FUNCTION_BLOCK FB_ATMTest EXTENDS FB_TestSuite
VAR
    (* Caller-owned axis, persistent storage, and Y motor.
       In a real PRG the AxisRef would come from MAIN.Mxx. *)
    axRef    : AXIS_REF;
    fbPDS    : LCLS_Tc_DevAbs.FB_PersistentDataStorage;

    (* FB_ATM is single-axis (nActiveMotorCount := 1), so only slot 1
       holds a real motor. aiMotionStage is sized to
       MotionConstants.MAX_STATE_MOTORS to match FB_ATM.FB_Init's
       fixed-size signature; slots 2-4 default-init to a nil interface
       and are never touched. *)
    fbMotorY : FB_MotionStageNC(AxisRef := axRef, iPersistentDataStorage := fbPDS, sName := 'Y');
    aiMotionStage : ARRAY[1..MotionConstants.MAX_STATE_MOTORS] OF I_MotionStage := [fbMotorY];

    {attribute 'pytmc' := '
        pv: MMS
        astPositionState.array: 1..6
    '}
    astPositionState : ARRAY[1..MotionConstants.MAX_STATE_MOTORS]
                         OF ARRAY[1..GeneralConstants.MAX_STATES] OF ST_PositionState;

    fbFFHWO    : FB_HardwareFFOutput;
    fbArbiter  : FB_Arbiter(1);
    fbSubSysIO : FB_DummyArbIO;

    sDeviceName    : STRING := 'TST:ATM';
    sTransitionKey : STRING := 'TST:ATM-TRANSITION';

    fbATM : FB_ATM(
        aiMotionStage         := aiMotionStage,
        astPositionState      := astPositionState,
        fbFFHWO               := fbFFHWO,
        fbArbiter             := fbArbiter,
        sDeviceName           := sDeviceName,
        sTransitionKey        := sTransitionKey,
        bEnableBeamParams     := TRUE,
        bEnablePositionLimits := TRUE,
        bReadDBNow            := TRUE
    );

    (* Per-install PMPS-side state config (caller-owned). Mirrors what
       a real PRG_xxL0_ATM would declare. stDefault is the caller-owned
       baseline template that FB_CC_StatePMPSConfig's inner FB_StateSetup
       preloads from; fbATM subsequently overrides per-state sName and
       fDelta via its own FB_CC_DeviceStateDefaults array. *)
    stDefault : ST_PositionState := (
        bMoveOk       := TRUE,
        bValid        := TRUE,
        bUseRawCounts := FALSE
    );

    afbStatePMPS : ARRAY[1..6] OF FB_CC_StatePMPSConfig[
        (stPositionState := astPositionState[1][E_ATM_States.OUT],
         stDefault       := stDefault,
         fPosition       := 10,
         sPmpsState      := 'TST:ATM-OUT'),
        (stPositionState := astPositionState[1][E_ATM_States.TARGET1],
         stDefault       := stDefault,
         fPosition       := 20,
         sPmpsState      := 'TST:ATM-TARGET1'),
        (stPositionState := astPositionState[1][E_ATM_States.TARGET2],
         stDefault       := stDefault,
         fPosition       := 30,
         sPmpsState      := 'TST:ATM-TARGET2'),
        (stPositionState := astPositionState[1][E_ATM_States.TARGET3],
         stDefault       := stDefault,
         fPosition       := 40,
         sPmpsState      := 'TST:ATM-TARGET3'),
        (stPositionState := astPositionState[1][E_ATM_States.TARGET4],
         stDefault       := stDefault,
         fPosition       := 50,
         sPmpsState      := 'TST:ATM-TARGET4'),
        (stPositionState := astPositionState[1][E_ATM_States.TARGET5],
         stDefault       := stDefault,
         fPosition       := 60,
         sPmpsState      := 'TST:ATM-TARGET5')
    ];

    bFirstScan : BOOL := TRUE;
    i          : UINT;
END_VAR

(* Fake PMPS handling. *)
fbSubSysIO(
    LA  := fbArbiter,
    FFO := fbFFHWO
);

(* Caller-side PMPS configurators write each slot once in
   FB_CC_StatePMPSConfig.CallAfterInit; no cyclic tick. *)

(* One-shot motor setup + initial caller-owned enables. Limits,
   brake/enable modes, home cmd, user/hardware enables, default
   velocity; skip NC param restore. *)
IF bFirstScan THEN
    fbMotorY.SetModeEnableLimits(
        LimBackward    := TRUE,
        LimForward     := TRUE,
        HomeEnable     := FALSE,
        BrakeMode      := E_StageBrakeMode.IF_ENABLED,
        EnableMode     := E_StageEnableMode.DURING_MOTION,
        HomeMode       := E_EpicsHomeCmd.LOW_LIMIT,
        UserEnable     := TRUE,
        HardwareEnable := TRUE
    );
    fbMotorY.SetVelocity(Velocity := 15.5);
    fbMotorY.RestoreMotionParams      := FALSE;
    fbMotorY.DoNotRestoreNcParameters := TRUE;

    bFirstScan := FALSE;
END_IF

fbPDS();
fbMotorY();
fbATM();

TestStateMove();
TestTempFFO();

METHOD SetATMTemp
VAR_INPUT
    iTempC : INT;
END_VAR
VAR
    ptr : POINTER TO INT;
END_VAR
ptr  := ADR(fbATM.fbTempSensor1.iRaw);
ptr^ := iTempC * 10;
END_METHOD

(*
    Smoke test for ATM state-move wiring. Walks OUT then TARGET1 and
    asserts each lands within fTolerance of the configured fPosition.
    Mirrors FB_REFTest: stageReady gate up front, NOT bMoving +
    position-tolerance check per state, 60s watchdog, on timeout
    AssertTrue(FALSE, ...) with the current step and observed
    position. Two moves is enough to exercise the FB wiring; the
    motion stack itself is covered by the
    lcls-twincat-motion-abstraction test suite.
*)
METHOD TestStateMove
VAR_INST
    tonTimer  : TON;
    nTestStep : INT := 0;
    fObserved : LREAL;
END_VAR
VAR CONSTANT
    fTolerance : LREAL := 2.0;
END_VAR
TEST('TestATMStateMove');

tonTimer(IN := TRUE, PT := T#60s);
fObserved := fbMotorY.stMotionStatus.fActPosition;

CASE nTestStep OF
    0:
        IF fbMotorY.stMotionStatus.bStageReady
           AND NOT fbMotorY.stMotionStatus.bError THEN
            fbATM.eEnumSet := E_ATM_States.OUT;
            nTestStep      := 1;
        END_IF
    1:
        (* OUT is configured at fPosition := 10 in afbStatePMPS[1]. *)
        IF fbATM.eEnumGet = E_ATM_States.OUT
           AND NOT fbMotorY.stMotionStatus.bMoving
           AND ABS(fObserved - 10.0) <= fTolerance THEN
            fbATM.eEnumSet := E_ATM_States.TARGET1;
            nTestStep      := 2;
        END_IF
    2:
        (* TARGET1 is configured at fPosition := 20 in afbStatePMPS[2]. *)
        IF fbATM.eEnumGet = E_ATM_States.TARGET1
           AND NOT fbMotorY.stMotionStatus.bMoving
           AND ABS(fObserved - 20.0) <= fTolerance THEN
            AssertTrue(
                Condition := TRUE,
                Message   := 'TestATMStateMove: OUT then TARGET1 reached within tolerance');
            nTestStep := 3;
        END_IF
END_CASE

IF nTestStep = 3 THEN
    TEST_FINISHED();
ELSIF tonTimer.Q THEN
    AssertTrue(
        Condition := FALSE,
        Message   := CONCAT(
            CONCAT(
                CONCAT('TestATMStateMove: timed out at step ', TO_STRING(nTestStep)),
                CONCAT(', eEnumGet=', TO_STRING(TO_UDINT(fbATM.eEnumGet)))),
            CONCAT(', fActPos=', TO_STRING(fObserved))));
    TEST_FINISHED();
END_IF
END_METHOD

METHOD TestTempFFO
VAR_INST
    tonTimer    : TON;
    nStep       : UINT := 0;
    bOutChecked : BOOL := FALSE;
    bInChecked  : BOOL := FALSE;
END_VAR
VAR CONSTANT
    nLastStep : UINT := 3;
END_VAR

(* Do we fault at the correct times?
   Parasitically depends on state move test. *)
TEST('TestATMTempFFO');

(* Prepare a timeout *)
tonTimer(IN := TRUE, PT := T#10s);

CASE nStep OF
    0:
        (* Set the thermocouple temperature to crazy high number. *)
        SetATMTemp(100);
        nStep := nStep + 1;
    1:
        (* Wait till we see "OUT" state and one other state (OUT
           should be no fault). *)
        IF fbATM.eEnumGet = E_ATM_States.OUT THEN
            AssertTrue(
                fbATM.fbTempSensor1.FFO.i_xOK,
                'Faulted even in out position!'
            );
            bOutChecked := TRUE;
        ELSIF fbATM.eEnumGet <> E_ATM_States.Unknown THEN
            AssertFalse(
                fbATM.fbTempSensor1.FFO.i_xOK,
                'No fault even for an in position!'
            );
            bInChecked := TRUE;
        END_IF
        IF bOutChecked AND bInChecked THEN
            nStep := nStep + 1;
        END_IF
    2:
        (* Set the thermocouple temperature to low again. *)
        SetATMTemp(0);
        nStep := nStep + 1;
    3:
        AssertTrue(
            fbATM.fbTempSensor1.FFO.i_xOK,
            'Faulted even with low temp!'
        );
        nStep := nStep + 1;
END_CASE

IF tonTimer.Q OR nStep > nLastStep THEN
    AssertFalse(tonTimer.Q, 'Timeout in ATM temp FFO test');
    TEST_FINISHED();
END_IF
END_METHOD

END_FUNCTION_BLOCK

(* stored: Version 1.1.0.1
   POU FB_ATMTest: Id {7b7c37ef-d7db-42bb-948f-8b077a7ccce5}, SpecialFunc None
   Method SetATMTemp: Id {7b7c37f0-d7db-42bb-948f-8b077a7ccce6}
   Method TestStateMove: Id {7b7c37f1-d7db-42bb-948f-8b077a7ccce7}
   Method TestTempFFO: Id {7b7c37f2-d7db-42bb-948f-8b077a7ccce8} *)
